// TIA Portal V17 export
// export: Created 2025-06-26T07:49:57.6379942Z, ExportSetting WithDefaults, DisplayName Totally Integrated Automation Portal, DisplayVersion V17 Update 8, DisplayName TIA Portal Openness, DisplayVersion V17 Update 8, DisplayName TIA Portal Version Control Interface, DisplayVersion V17, DisplayName STEP 7 Professional, DisplayVersion V17 Update 8, DisplayName STEP 7 Safety, DisplayVersion V17 Update 6, DisplayName WinCC Advanced, DisplayVersion V17 Update 8
TYPE "FluidBasedLimits-STRUCT"
// stored: IsFailsafeCompliant false
   STRUCT
      T_HeatSourceTemperature_Max : Real;
      T_HeatSourceTemperature_Min : Real;
      T_HeatSinkTemperature_Max : Real;
      T_OilTemperature_Critical : Real := 140.0;
      T_OilSuperheat : Real := 8.0;
      T_CoolingSetpoint : Real := 110.0;
   END_STRUCT;
END_TYPE
